TYPE E_Typ_MOD :
(
	///no usage until yet
	Default := 0,
	Max_E_Typ_CYL
);
END_TYPE

(* stored: Version 1.1.0.1, ProductVersion 3.1.0.14
   DUT E_Typ_MOD: Id {996e7dfd-30bb-4433-87f2-b569c8ff5d7f} *)
